PROGRAM Alarm_Warring
VAR
//System_Bit
	Always_ON				:	BOOL	:=TRUE	;//상시 ON
	Always_OFF				:	BOOL	:=FALSE	;//상시 OFF	
END_VAR

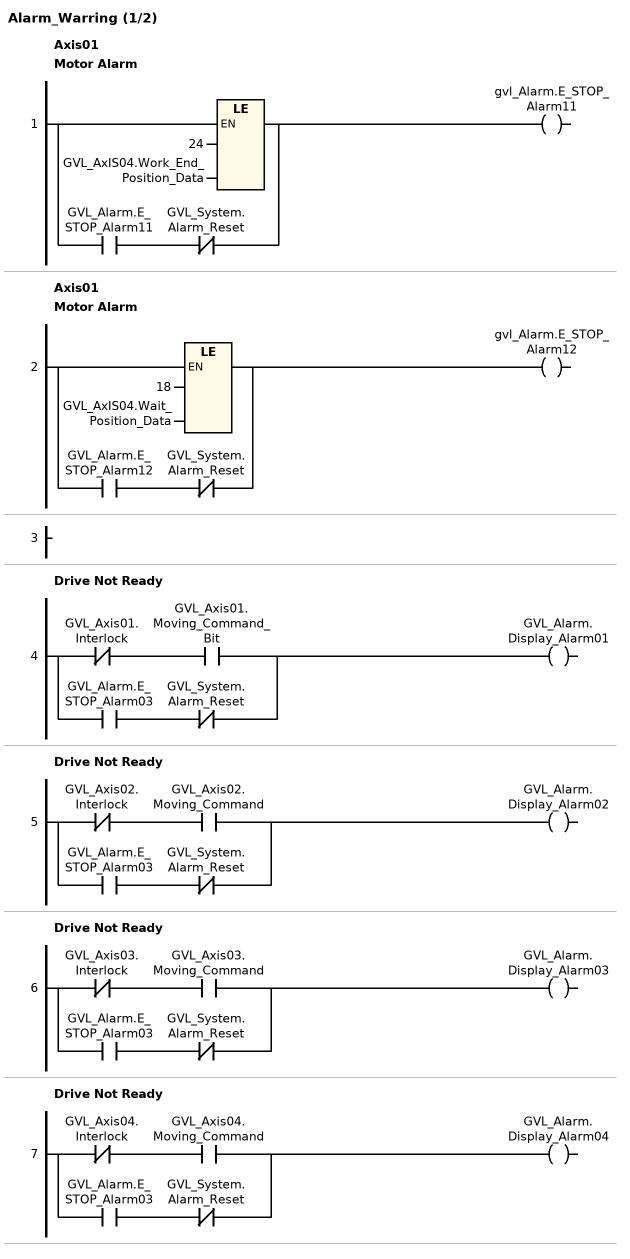
// NETWORK 1: Axis01 Motor Alarm
gvl_Alarm.E_STOP_Alarm11 := 24 <= GVL_AxIS04.Work_End_Position_Data OR GVL_Alarm.E_STOP_Alarm11 AND NOT GVL_System.Alarm_Reset;

// NETWORK 2: Axis01 Motor Alarm
gvl_Alarm.E_STOP_Alarm12 := 18 <= GVL_AxIS04.Wait_Position_Data OR GVL_Alarm.E_STOP_Alarm12 AND NOT GVL_System.Alarm_Reset;

// NETWORK 3

// NETWORK 4: Drive Not Ready
GVL_Alarm.Display_Alarm01 := NOT GVL_Axis01.Interlock AND GVL_Axis01.Moving_Command_Bit OR GVL_Alarm.E_STOP_Alarm03 AND NOT GVL_System.Alarm_Reset;

// NETWORK 5: Drive Not Ready
GVL_Alarm.Display_Alarm02 := NOT GVL_Axis02.Interlock AND GVL_Axis02.Moving_Command OR GVL_Alarm.E_STOP_Alarm03 AND NOT GVL_System.Alarm_Reset;

// NETWORK 6: Drive Not Ready
GVL_Alarm.Display_Alarm03 := NOT GVL_Axis03.Interlock AND GVL_Axis03.Moving_Command OR GVL_Alarm.E_STOP_Alarm03 AND NOT GVL_System.Alarm_Reset;

// NETWORK 7: Drive Not Ready
GVL_Alarm.Display_Alarm04 := NOT GVL_Axis04.Interlock AND GVL_Axis04.Moving_Command OR GVL_Alarm.E_STOP_Alarm03 AND NOT GVL_System.Alarm_Reset;

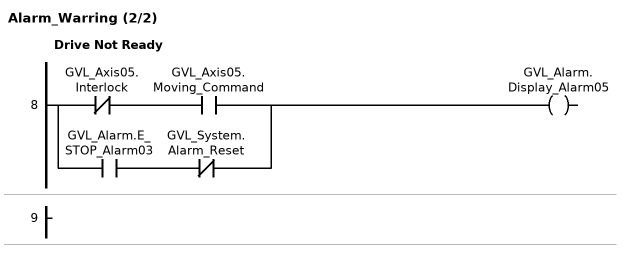
// NETWORK 8: Drive Not Ready
GVL_Alarm.Display_Alarm05 := NOT GVL_Axis05.Interlock AND GVL_Axis05.Moving_Command OR GVL_Alarm.E_STOP_Alarm03 AND NOT GVL_System.Alarm_Reset;

// NETWORK 9

END_PROGRAM

(* stored: Version 1.1.0.1, ProductVersion 3.1.4024.15
   POU Alarm_Warring: Id {a3c71ad0-95af-4ffa-b9d7-9d06ef845c64}, SpecialFunc None *)
